{attribute 'qualified_only'}
{attribute 'strict'}
{attribute 'to_string'}
TYPE e_Signal_Colors :
(
	ACTIVE_RED := 0,
	ACTIVE_YELLOW := 1,
	ACTIVE_GREEN := 2,
	PASSIVE_RED := 3,
	FLASHING_RED := 4
);
END_TYPE

(* stored: Version 1.1.0.1
   DUT e_Signal_Colors: Id {636b57e0-bcf9-43c6-aebd-664d8291dd79} *)
